// TIA Portal V18 export
// export: Created 2026-06-20T08:02:04.9898097Z, ExportSetting WithDefaults, DisplayName Totally Integrated Automation Portal, DisplayVersion V18, DisplayName TIA Portal Openness, DisplayVersion V18, DisplayName TIA Portal Version Control Interface, DisplayVersion V18, DisplayName STEP 7 Professional, DisplayVersion V18, DisplayName STEP 7 Safety, DisplayVersion V18, DisplayName WinCC Professional, DisplayVersion V18
ORGANIZATION_BLOCK "Main"   // OB1, LAD, ProgramCycle
TITLE = "Main Program Sweep (Cycle)"
{ S7_Optimized_Access := 'TRUE' }
VERSION : 0.1
// stored: AutoNumber true, IsIECCheckEnabled false, SetENOAutomatically false
   VAR_INPUT
      Initial_Call : Bool;   // Initial call of this OB
      Remanence : Bool;   // =True, if remanent data are available
   END_VAR
BEGIN

REGION Network 1: Clock 1Hz Edge Detection
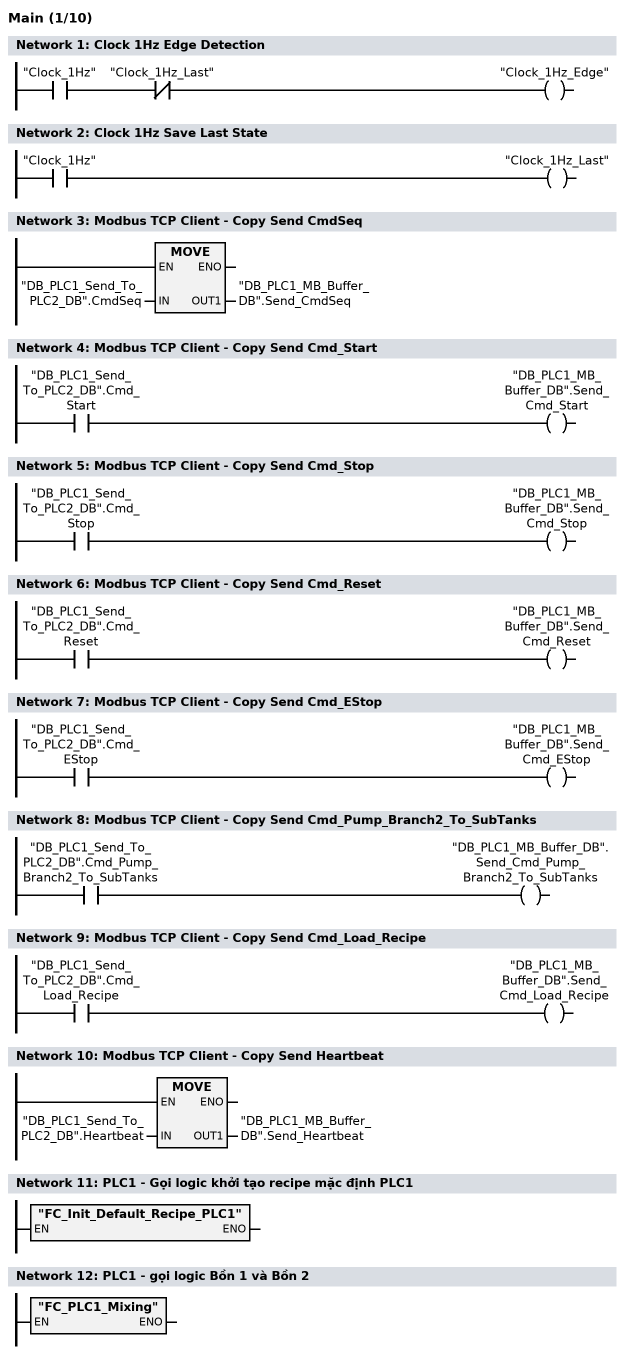
   RUNG wire#powerrail
      Contact( "Clock_1Hz" )
      I_Contact( "Clock_1Hz_Last" )
      Coil( "Clock_1Hz_Edge" )
   END_RUNG
   // the same network as SCL:
   "Clock_1Hz_Edge" := "Clock_1Hz" AND NOT "Clock_1Hz_Last";
END_REGION

REGION Network 2: Clock 1Hz Save Last State
   RUNG wire#powerrail
      Contact( "Clock_1Hz" )
      Coil( "Clock_1Hz_Last" )
   END_RUNG
   // the same network as SCL:
   "Clock_1Hz_Last" := "Clock_1Hz";
END_REGION

REGION Network 3: Modbus TCP Client - Copy Send CmdSeq
   RUNG wire#powerrail
      { S7_GenerateENO := "TRUE" } Move(in := "DB_PLC1_Send_To_PLC2_DB".CmdSeq, out1 => "DB_PLC1_MB_Buffer_DB".Send_CmdSeq)
   END_RUNG
   // the same network as SCL:
   "DB_PLC1_MB_Buffer_DB".Send_CmdSeq := "DB_PLC1_Send_To_PLC2_DB".CmdSeq;
END_REGION

REGION Network 4: Modbus TCP Client - Copy Send Cmd_Start
   RUNG wire#powerrail
      Contact( "DB_PLC1_Send_To_PLC2_DB".Cmd_Start )
      Coil( "DB_PLC1_MB_Buffer_DB".Send_Cmd_Start )
   END_RUNG
   // the same network as SCL:
   "DB_PLC1_MB_Buffer_DB".Send_Cmd_Start := "DB_PLC1_Send_To_PLC2_DB".Cmd_Start;
END_REGION

REGION Network 5: Modbus TCP Client - Copy Send Cmd_Stop
   RUNG wire#powerrail
      Contact( "DB_PLC1_Send_To_PLC2_DB".Cmd_Stop )
      Coil( "DB_PLC1_MB_Buffer_DB".Send_Cmd_Stop )
   END_RUNG
   // the same network as SCL:
   "DB_PLC1_MB_Buffer_DB".Send_Cmd_Stop := "DB_PLC1_Send_To_PLC2_DB".Cmd_Stop;
END_REGION

REGION Network 6: Modbus TCP Client - Copy Send Cmd_Reset
   RUNG wire#powerrail
      Contact( "DB_PLC1_Send_To_PLC2_DB".Cmd_Reset )
      Coil( "DB_PLC1_MB_Buffer_DB".Send_Cmd_Reset )
   END_RUNG
   // the same network as SCL:
   "DB_PLC1_MB_Buffer_DB".Send_Cmd_Reset := "DB_PLC1_Send_To_PLC2_DB".Cmd_Reset;
END_REGION

REGION Network 7: Modbus TCP Client - Copy Send Cmd_EStop
   RUNG wire#powerrail
      Contact( "DB_PLC1_Send_To_PLC2_DB".Cmd_EStop )
      Coil( "DB_PLC1_MB_Buffer_DB".Send_Cmd_EStop )
   END_RUNG
   // the same network as SCL:
   "DB_PLC1_MB_Buffer_DB".Send_Cmd_EStop := "DB_PLC1_Send_To_PLC2_DB".Cmd_EStop;
END_REGION

REGION Network 8: Modbus TCP Client - Copy Send Cmd_Pump_Branch2_To_SubTanks
   RUNG wire#powerrail
      Contact( "DB_PLC1_Send_To_PLC2_DB".Cmd_Pump_Branch2_To_SubTanks )
      Coil( "DB_PLC1_MB_Buffer_DB".Send_Cmd_Pump_Branch2_To_SubTanks )
   END_RUNG
   // the same network as SCL:
   "DB_PLC1_MB_Buffer_DB".Send_Cmd_Pump_Branch2_To_SubTanks := "DB_PLC1_Send_To_PLC2_DB".Cmd_Pump_Branch2_To_SubTanks;
END_REGION

REGION Network 9: Modbus TCP Client - Copy Send Cmd_Load_Recipe
   RUNG wire#powerrail
      Contact( "DB_PLC1_Send_To_PLC2_DB".Cmd_Load_Recipe )
      Coil( "DB_PLC1_MB_Buffer_DB".Send_Cmd_Load_Recipe )
   END_RUNG
   // the same network as SCL:
   "DB_PLC1_MB_Buffer_DB".Send_Cmd_Load_Recipe := "DB_PLC1_Send_To_PLC2_DB".Cmd_Load_Recipe;
END_REGION

REGION Network 10: Modbus TCP Client - Copy Send Heartbeat
   RUNG wire#powerrail
      { S7_GenerateENO := "TRUE" } Move(in := "DB_PLC1_Send_To_PLC2_DB".Heartbeat, out1 => "DB_PLC1_MB_Buffer_DB".Send_Heartbeat)
   END_RUNG
   // the same network as SCL:
   "DB_PLC1_MB_Buffer_DB".Send_Heartbeat := "DB_PLC1_Send_To_PLC2_DB".Heartbeat;
END_REGION

REGION Network 11: PLC1 - Gọi logic khởi tạo recipe mặc định PLC1
   RUNG wire#powerrail
      "FC_Init_Default_Recipe_PLC1"()
   END_RUNG
   // the same network as SCL:
   "FC_Init_Default_Recipe_PLC1"();
END_REGION

REGION Network 12: PLC1 - gọi logic Bồn 1 và Bồn 2
   RUNG wire#powerrail
      "FC_PLC1_Mixing"()
   END_RUNG
   // the same network as SCL:
   "FC_PLC1_Mixing"();
END_REGION

REGION Network 13: PLC1 - gọi logic bồn chứa và lọc thành phẩm
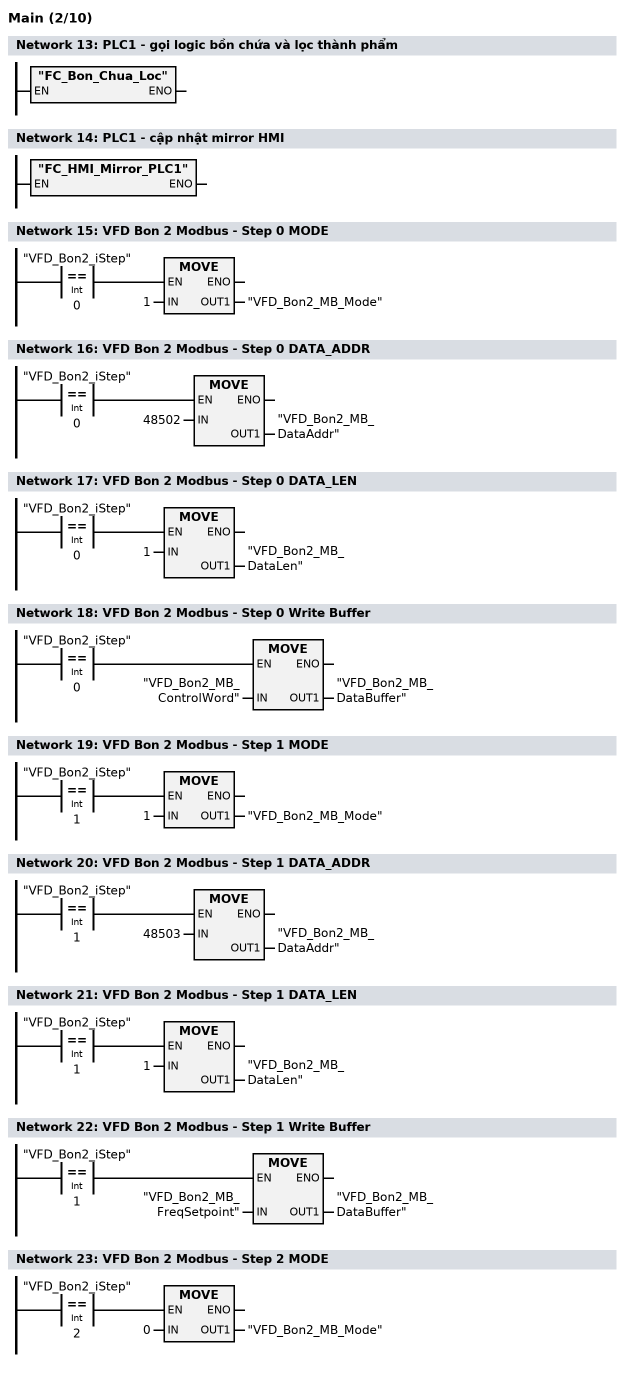
   RUNG wire#powerrail
      "FC_Bon_Chua_Loc"()
   END_RUNG
   // the same network as SCL:
   "FC_Bon_Chua_Loc"();
END_REGION

REGION Network 14: PLC1 - cập nhật mirror HMI
   RUNG wire#powerrail
      "FC_HMI_Mirror_PLC1"()
   END_RUNG
   // the same network as SCL:
   "FC_HMI_Mirror_PLC1"();
END_REGION

REGION Network 15: VFD Bon 2 Modbus - Step 0 MODE
   RUNG wire#powerrail
      { S7_Templates := "SrcType := Int" } EQ_Contact(in1 := "VFD_Bon2_iStep", in2 := 0)
      { S7_GenerateENO := "TRUE" } Move(in := 1, out1 => "VFD_Bon2_MB_Mode")
   END_RUNG
   // the same network as SCL:
   IF "VFD_Bon2_iStep" = 0 THEN "VFD_Bon2_MB_Mode" := 1; END_IF;
END_REGION

REGION Network 16: VFD Bon 2 Modbus - Step 0 DATA_ADDR
   RUNG wire#powerrail
      { S7_Templates := "SrcType := Int" } EQ_Contact(in1 := "VFD_Bon2_iStep", in2 := 0)
      { S7_GenerateENO := "TRUE" } Move(in := 48502, out1 => "VFD_Bon2_MB_DataAddr")
   END_RUNG
   // the same network as SCL:
   IF "VFD_Bon2_iStep" = 0 THEN "VFD_Bon2_MB_DataAddr" := 48502; END_IF;
END_REGION

REGION Network 17: VFD Bon 2 Modbus - Step 0 DATA_LEN
   RUNG wire#powerrail
      { S7_Templates := "SrcType := Int" } EQ_Contact(in1 := "VFD_Bon2_iStep", in2 := 0)
      { S7_GenerateENO := "TRUE" } Move(in := 1, out1 => "VFD_Bon2_MB_DataLen")
   END_RUNG
   // the same network as SCL:
   IF "VFD_Bon2_iStep" = 0 THEN "VFD_Bon2_MB_DataLen" := 1; END_IF;
END_REGION

REGION Network 18: VFD Bon 2 Modbus - Step 0 Write Buffer
   RUNG wire#powerrail
      { S7_Templates := "SrcType := Int" } EQ_Contact(in1 := "VFD_Bon2_iStep", in2 := 0)
      { S7_GenerateENO := "TRUE" } Move(in := "VFD_Bon2_MB_ControlWord", out1 => "VFD_Bon2_MB_DataBuffer")
   END_RUNG
   // the same network as SCL:
   IF "VFD_Bon2_iStep" = 0 THEN "VFD_Bon2_MB_DataBuffer" := "VFD_Bon2_MB_ControlWord"; END_IF;
END_REGION

REGION Network 19: VFD Bon 2 Modbus - Step 1 MODE
   RUNG wire#powerrail
      { S7_Templates := "SrcType := Int" } EQ_Contact(in1 := "VFD_Bon2_iStep", in2 := 1)
      { S7_GenerateENO := "TRUE" } Move(in := 1, out1 => "VFD_Bon2_MB_Mode")
   END_RUNG
   // the same network as SCL:
   IF "VFD_Bon2_iStep" = 1 THEN "VFD_Bon2_MB_Mode" := 1; END_IF;
END_REGION

REGION Network 20: VFD Bon 2 Modbus - Step 1 DATA_ADDR
   RUNG wire#powerrail
      { S7_Templates := "SrcType := Int" } EQ_Contact(in1 := "VFD_Bon2_iStep", in2 := 1)
      { S7_GenerateENO := "TRUE" } Move(in := 48503, out1 => "VFD_Bon2_MB_DataAddr")
   END_RUNG
   // the same network as SCL:
   IF "VFD_Bon2_iStep" = 1 THEN "VFD_Bon2_MB_DataAddr" := 48503; END_IF;
END_REGION

REGION Network 21: VFD Bon 2 Modbus - Step 1 DATA_LEN
   RUNG wire#powerrail
      { S7_Templates := "SrcType := Int" } EQ_Contact(in1 := "VFD_Bon2_iStep", in2 := 1)
      { S7_GenerateENO := "TRUE" } Move(in := 1, out1 => "VFD_Bon2_MB_DataLen")
   END_RUNG
   // the same network as SCL:
   IF "VFD_Bon2_iStep" = 1 THEN "VFD_Bon2_MB_DataLen" := 1; END_IF;
END_REGION

REGION Network 22: VFD Bon 2 Modbus - Step 1 Write Buffer
   RUNG wire#powerrail
      { S7_Templates := "SrcType := Int" } EQ_Contact(in1 := "VFD_Bon2_iStep", in2 := 1)
      { S7_GenerateENO := "TRUE" } Move(in := "VFD_Bon2_MB_FreqSetpoint", out1 => "VFD_Bon2_MB_DataBuffer")
   END_RUNG
   // the same network as SCL:
   IF "VFD_Bon2_iStep" = 1 THEN "VFD_Bon2_MB_DataBuffer" := "VFD_Bon2_MB_FreqSetpoint"; END_IF;
END_REGION

REGION Network 23: VFD Bon 2 Modbus - Step 2 MODE
   RUNG wire#powerrail
      { S7_Templates := "SrcType := Int" } EQ_Contact(in1 := "VFD_Bon2_iStep", in2 := 2)
      { S7_GenerateENO := "TRUE" } Move(in := 0, out1 => "VFD_Bon2_MB_Mode")
   END_RUNG
   // the same network as SCL:
   IF "VFD_Bon2_iStep" = 2 THEN "VFD_Bon2_MB_Mode" := 0; END_IF;
END_REGION

REGION Network 24: VFD Bon 2 Modbus - Step 2 DATA_ADDR
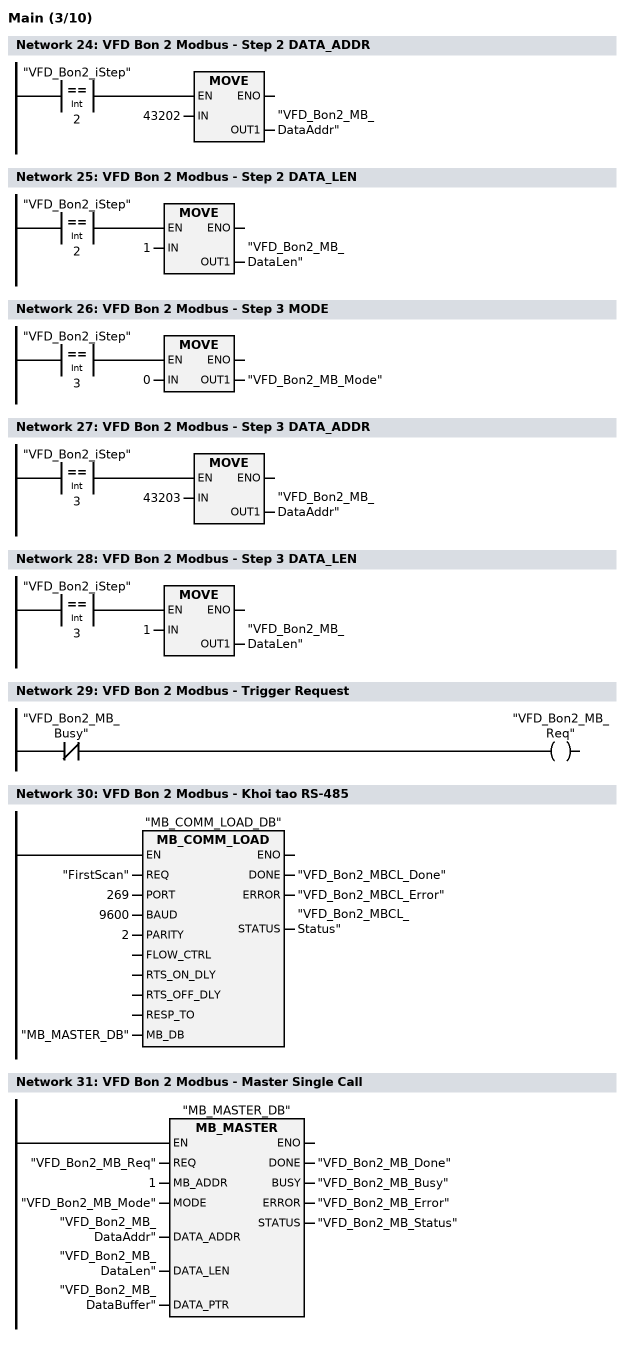
   RUNG wire#powerrail
      { S7_Templates := "SrcType := Int" } EQ_Contact(in1 := "VFD_Bon2_iStep", in2 := 2)
      { S7_GenerateENO := "TRUE" } Move(in := 43202, out1 => "VFD_Bon2_MB_DataAddr")
   END_RUNG
   // the same network as SCL:
   IF "VFD_Bon2_iStep" = 2 THEN "VFD_Bon2_MB_DataAddr" := 43202; END_IF;
END_REGION

REGION Network 25: VFD Bon 2 Modbus - Step 2 DATA_LEN
   RUNG wire#powerrail
      { S7_Templates := "SrcType := Int" } EQ_Contact(in1 := "VFD_Bon2_iStep", in2 := 2)
      { S7_GenerateENO := "TRUE" } Move(in := 1, out1 => "VFD_Bon2_MB_DataLen")
   END_RUNG
   // the same network as SCL:
   IF "VFD_Bon2_iStep" = 2 THEN "VFD_Bon2_MB_DataLen" := 1; END_IF;
END_REGION

REGION Network 26: VFD Bon 2 Modbus - Step 3 MODE
   RUNG wire#powerrail
      { S7_Templates := "SrcType := Int" } EQ_Contact(in1 := "VFD_Bon2_iStep", in2 := 3)
      { S7_GenerateENO := "TRUE" } Move(in := 0, out1 => "VFD_Bon2_MB_Mode")
   END_RUNG
   // the same network as SCL:
   IF "VFD_Bon2_iStep" = 3 THEN "VFD_Bon2_MB_Mode" := 0; END_IF;
END_REGION

REGION Network 27: VFD Bon 2 Modbus - Step 3 DATA_ADDR
   RUNG wire#powerrail
      { S7_Templates := "SrcType := Int" } EQ_Contact(in1 := "VFD_Bon2_iStep", in2 := 3)
      { S7_GenerateENO := "TRUE" } Move(in := 43203, out1 => "VFD_Bon2_MB_DataAddr")
   END_RUNG
   // the same network as SCL:
   IF "VFD_Bon2_iStep" = 3 THEN "VFD_Bon2_MB_DataAddr" := 43203; END_IF;
END_REGION

REGION Network 28: VFD Bon 2 Modbus - Step 3 DATA_LEN
   RUNG wire#powerrail
      { S7_Templates := "SrcType := Int" } EQ_Contact(in1 := "VFD_Bon2_iStep", in2 := 3)
      { S7_GenerateENO := "TRUE" } Move(in := 1, out1 => "VFD_Bon2_MB_DataLen")
   END_RUNG
   // the same network as SCL:
   IF "VFD_Bon2_iStep" = 3 THEN "VFD_Bon2_MB_DataLen" := 1; END_IF;
END_REGION

REGION Network 29: VFD Bon 2 Modbus - Trigger Request
   RUNG wire#powerrail
      I_Contact( "VFD_Bon2_MB_Busy" )
      Coil( "VFD_Bon2_MB_Req" )
   END_RUNG
   // the same network as SCL:
   "VFD_Bon2_MB_Req" := NOT "VFD_Bon2_MB_Busy";
END_REGION

REGION Network 30: VFD Bon 2 Modbus - Khoi tao RS-485
   RUNG wire#powerrail
      "MB_COMM_LOAD_DB".MB_COMM_LOAD(REQ := "FirstScan", PORT := 269, BAUD := 9600, PARITY := 2, FLOW_CTRL :=, RTS_ON_DLY :=, RTS_OFF_DLY :=, RESP_TO :=, MB_DB := "MB_MASTER_DB", DONE => "VFD_Bon2_MBCL_Done", ERROR => "VFD_Bon2_MBCL_Error", STATUS => "VFD_Bon2_MBCL_Status")
   END_RUNG
   // the same network as SCL:
   "MB_COMM_LOAD_DB"(REQ := "FirstScan",   // MB_COMM_LOAD
                     PORT := 269,
                     BAUD := 9600,
                     PARITY := 2,
                     MB_DB := "MB_MASTER_DB",
                     DONE => "VFD_Bon2_MBCL_Done",
                     ERROR => "VFD_Bon2_MBCL_Error",
                     STATUS => "VFD_Bon2_MBCL_Status");
END_REGION

REGION Network 31: VFD Bon 2 Modbus - Master Single Call
   RUNG wire#powerrail
      "MB_MASTER_DB".MB_MASTER(REQ := "VFD_Bon2_MB_Req", MB_ADDR := 1, MODE := "VFD_Bon2_MB_Mode", DATA_ADDR := "VFD_Bon2_MB_DataAddr", DATA_LEN := "VFD_Bon2_MB_DataLen", DATA_PTR := "VFD_Bon2_MB_DataBuffer", DONE => "VFD_Bon2_MB_Done", BUSY => "VFD_Bon2_MB_Busy", ERROR => "VFD_Bon2_MB_Error", STATUS => "VFD_Bon2_MB_Status")
   END_RUNG
   // the same network as SCL:
   "MB_MASTER_DB"(REQ := "VFD_Bon2_MB_Req",   // MB_MASTER
                  MB_ADDR := 1,
                  MODE := "VFD_Bon2_MB_Mode",
                  DATA_ADDR := "VFD_Bon2_MB_DataAddr",
                  DATA_LEN := "VFD_Bon2_MB_DataLen",
                  DATA_PTR := "VFD_Bon2_MB_DataBuffer",
                  DONE => "VFD_Bon2_MB_Done",
                  BUSY => "VFD_Bon2_MB_Busy",
                  ERROR => "VFD_Bon2_MB_Error",
                  STATUS => "VFD_Bon2_MB_Status");
END_REGION

REGION Network 32: VFD Bon 2 Modbus - Read Step 2 Buffer Copy
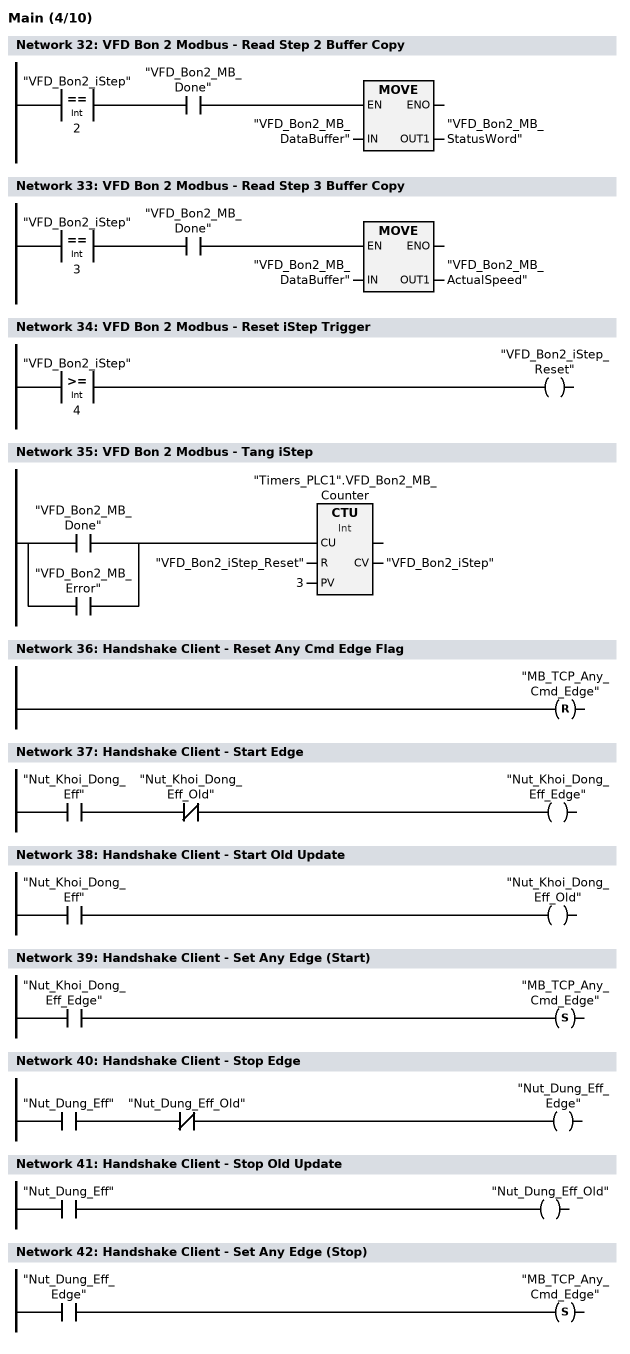
   RUNG wire#powerrail
      { S7_Templates := "SrcType := Int" } EQ_Contact(in1 := "VFD_Bon2_iStep", in2 := 2)
      Contact( "VFD_Bon2_MB_Done" )
      { S7_GenerateENO := "TRUE" } Move(in := "VFD_Bon2_MB_DataBuffer", out1 => "VFD_Bon2_MB_StatusWord")
   END_RUNG
   // the same network as SCL:
   IF ("VFD_Bon2_iStep" = 2) AND "VFD_Bon2_MB_Done" THEN
       "VFD_Bon2_MB_StatusWord" := "VFD_Bon2_MB_DataBuffer";
   END_IF;
END_REGION

REGION Network 33: VFD Bon 2 Modbus - Read Step 3 Buffer Copy
   RUNG wire#powerrail
      { S7_Templates := "SrcType := Int" } EQ_Contact(in1 := "VFD_Bon2_iStep", in2 := 3)
      Contact( "VFD_Bon2_MB_Done" )
      { S7_GenerateENO := "TRUE" } Move(in := "VFD_Bon2_MB_DataBuffer", out1 => "VFD_Bon2_MB_ActualSpeed")
   END_RUNG
   // the same network as SCL:
   IF ("VFD_Bon2_iStep" = 3) AND "VFD_Bon2_MB_Done" THEN
       "VFD_Bon2_MB_ActualSpeed" := "VFD_Bon2_MB_DataBuffer";
   END_IF;
END_REGION

REGION Network 34: VFD Bon 2 Modbus - Reset iStep Trigger
   RUNG wire#powerrail
      { S7_Templates := "SrcType := Int" } GE_Contact(in1 := "VFD_Bon2_iStep", in2 := 4)
      Coil( "VFD_Bon2_iStep_Reset" )
   END_RUNG
   // the same network as SCL:
   "VFD_Bon2_iStep_Reset" := "VFD_Bon2_iStep" >= 4;
END_REGION

REGION Network 35: VFD Bon 2 Modbus - Tang iStep
   RUNG wire#powerrail
      Contact( "VFD_Bon2_MB_Done" )
      wire#w1
      { S7_Templates := "value_type := Int" } "Timers_PLC1".VFD_Bon2_MB_Counter.CTU(r := "VFD_Bon2_iStep_Reset", pv := 3, cv => "VFD_Bon2_iStep")
   END_RUNG
   RUNG wire#powerrail
      Contact( "VFD_Bon2_MB_Error" )
   END_RUNG wire#w1
   // the same network as SCL:
   "Timers_PLC1".VFD_Bon2_MB_Counter.CTU(CU := "VFD_Bon2_MB_Done" OR "VFD_Bon2_MB_Error",
                           R := "VFD_Bon2_iStep_Reset",
                           PV := 3,
                           CV => "VFD_Bon2_iStep");
END_REGION

REGION Network 36: Handshake Client - Reset Any Cmd Edge Flag
   RUNG wire#powerrail
      R_Coil( "MB_TCP_Any_Cmd_Edge" )
   END_RUNG
   // the same network as SCL:
   "MB_TCP_Any_Cmd_Edge" := FALSE;
END_REGION

REGION Network 37: Handshake Client - Start Edge
   RUNG wire#powerrail
      Contact( "Nut_Khoi_Dong_Eff" )
      I_Contact( "Nut_Khoi_Dong_Eff_Old" )
      Coil( "Nut_Khoi_Dong_Eff_Edge" )
   END_RUNG
   // the same network as SCL:
   "Nut_Khoi_Dong_Eff_Edge" := "Nut_Khoi_Dong_Eff" AND NOT "Nut_Khoi_Dong_Eff_Old";
END_REGION

REGION Network 38: Handshake Client - Start Old Update
   RUNG wire#powerrail
      Contact( "Nut_Khoi_Dong_Eff" )
      Coil( "Nut_Khoi_Dong_Eff_Old" )
   END_RUNG
   // the same network as SCL:
   "Nut_Khoi_Dong_Eff_Old" := "Nut_Khoi_Dong_Eff";
END_REGION

REGION Network 39: Handshake Client - Set Any Edge (Start)
   RUNG wire#powerrail
      Contact( "Nut_Khoi_Dong_Eff_Edge" )
      S_Coil( "MB_TCP_Any_Cmd_Edge" )
   END_RUNG
   // the same network as SCL:
   IF "Nut_Khoi_Dong_Eff_Edge" THEN "MB_TCP_Any_Cmd_Edge" := TRUE; END_IF;
END_REGION

REGION Network 40: Handshake Client - Stop Edge
   RUNG wire#powerrail
      Contact( "Nut_Dung_Eff" )
      I_Contact( "Nut_Dung_Eff_Old" )
      Coil( "Nut_Dung_Eff_Edge" )
   END_RUNG
   // the same network as SCL:
   "Nut_Dung_Eff_Edge" := "Nut_Dung_Eff" AND NOT "Nut_Dung_Eff_Old";
END_REGION

REGION Network 41: Handshake Client - Stop Old Update
   RUNG wire#powerrail
      Contact( "Nut_Dung_Eff" )
      Coil( "Nut_Dung_Eff_Old" )
   END_RUNG
   // the same network as SCL:
   "Nut_Dung_Eff_Old" := "Nut_Dung_Eff";
END_REGION

REGION Network 42: Handshake Client - Set Any Edge (Stop)
   RUNG wire#powerrail
      Contact( "Nut_Dung_Eff_Edge" )
      S_Coil( "MB_TCP_Any_Cmd_Edge" )
   END_RUNG
   // the same network as SCL:
   IF "Nut_Dung_Eff_Edge" THEN "MB_TCP_Any_Cmd_Edge" := TRUE; END_IF;
END_REGION

REGION Network 43: Handshake Client - Reset Edge
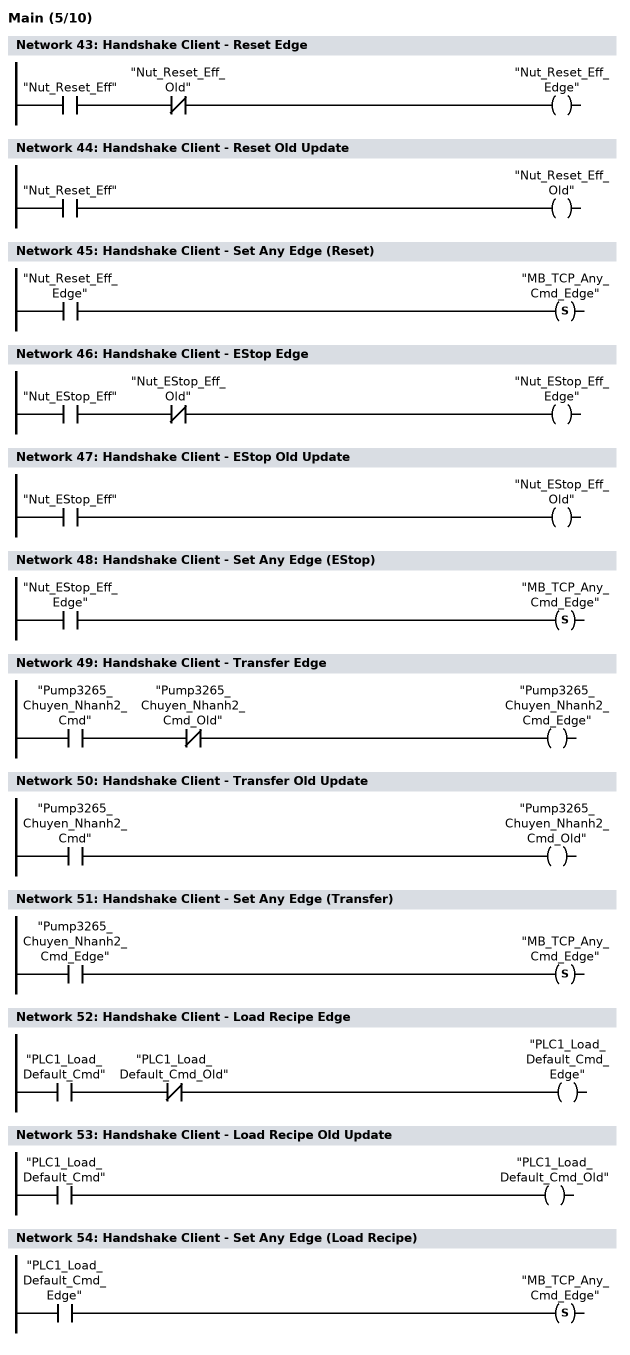
   RUNG wire#powerrail
      Contact( "Nut_Reset_Eff" )
      I_Contact( "Nut_Reset_Eff_Old" )
      Coil( "Nut_Reset_Eff_Edge" )
   END_RUNG
   // the same network as SCL:
   "Nut_Reset_Eff_Edge" := "Nut_Reset_Eff" AND NOT "Nut_Reset_Eff_Old";
END_REGION

REGION Network 44: Handshake Client - Reset Old Update
   RUNG wire#powerrail
      Contact( "Nut_Reset_Eff" )
      Coil( "Nut_Reset_Eff_Old" )
   END_RUNG
   // the same network as SCL:
   "Nut_Reset_Eff_Old" := "Nut_Reset_Eff";
END_REGION

REGION Network 45: Handshake Client - Set Any Edge (Reset)
   RUNG wire#powerrail
      Contact( "Nut_Reset_Eff_Edge" )
      S_Coil( "MB_TCP_Any_Cmd_Edge" )
   END_RUNG
   // the same network as SCL:
   IF "Nut_Reset_Eff_Edge" THEN "MB_TCP_Any_Cmd_Edge" := TRUE; END_IF;
END_REGION

REGION Network 46: Handshake Client - EStop Edge
   RUNG wire#powerrail
      Contact( "Nut_EStop_Eff" )
      I_Contact( "Nut_EStop_Eff_Old" )
      Coil( "Nut_EStop_Eff_Edge" )
   END_RUNG
   // the same network as SCL:
   "Nut_EStop_Eff_Edge" := "Nut_EStop_Eff" AND NOT "Nut_EStop_Eff_Old";
END_REGION

REGION Network 47: Handshake Client - EStop Old Update
   RUNG wire#powerrail
      Contact( "Nut_EStop_Eff" )
      Coil( "Nut_EStop_Eff_Old" )
   END_RUNG
   // the same network as SCL:
   "Nut_EStop_Eff_Old" := "Nut_EStop_Eff";
END_REGION

REGION Network 48: Handshake Client - Set Any Edge (EStop)
   RUNG wire#powerrail
      Contact( "Nut_EStop_Eff_Edge" )
      S_Coil( "MB_TCP_Any_Cmd_Edge" )
   END_RUNG
   // the same network as SCL:
   IF "Nut_EStop_Eff_Edge" THEN "MB_TCP_Any_Cmd_Edge" := TRUE; END_IF;
END_REGION

REGION Network 49: Handshake Client - Transfer Edge
   RUNG wire#powerrail
      Contact( "Pump3265_Chuyen_Nhanh2_Cmd" )
      I_Contact( "Pump3265_Chuyen_Nhanh2_Cmd_Old" )
      Coil( "Pump3265_Chuyen_Nhanh2_Cmd_Edge" )
   END_RUNG
   // the same network as SCL:
   "Pump3265_Chuyen_Nhanh2_Cmd_Edge" := "Pump3265_Chuyen_Nhanh2_Cmd" AND NOT "Pump3265_Chuyen_Nhanh2_Cmd_Old";
END_REGION

REGION Network 50: Handshake Client - Transfer Old Update
   RUNG wire#powerrail
      Contact( "Pump3265_Chuyen_Nhanh2_Cmd" )
      Coil( "Pump3265_Chuyen_Nhanh2_Cmd_Old" )
   END_RUNG
   // the same network as SCL:
   "Pump3265_Chuyen_Nhanh2_Cmd_Old" := "Pump3265_Chuyen_Nhanh2_Cmd";
END_REGION

REGION Network 51: Handshake Client - Set Any Edge (Transfer)
   RUNG wire#powerrail
      Contact( "Pump3265_Chuyen_Nhanh2_Cmd_Edge" )
      S_Coil( "MB_TCP_Any_Cmd_Edge" )
   END_RUNG
   // the same network as SCL:
   IF "Pump3265_Chuyen_Nhanh2_Cmd_Edge" THEN "MB_TCP_Any_Cmd_Edge" := TRUE; END_IF;
END_REGION

REGION Network 52: Handshake Client - Load Recipe Edge
   RUNG wire#powerrail
      Contact( "PLC1_Load_Default_Cmd" )
      I_Contact( "PLC1_Load_Default_Cmd_Old" )
      Coil( "PLC1_Load_Default_Cmd_Edge" )
   END_RUNG
   // the same network as SCL:
   "PLC1_Load_Default_Cmd_Edge" := "PLC1_Load_Default_Cmd" AND NOT "PLC1_Load_Default_Cmd_Old";
END_REGION

REGION Network 53: Handshake Client - Load Recipe Old Update
   RUNG wire#powerrail
      Contact( "PLC1_Load_Default_Cmd" )
      Coil( "PLC1_Load_Default_Cmd_Old" )
   END_RUNG
   // the same network as SCL:
   "PLC1_Load_Default_Cmd_Old" := "PLC1_Load_Default_Cmd";
END_REGION

REGION Network 54: Handshake Client - Set Any Edge (Load Recipe)
   RUNG wire#powerrail
      Contact( "PLC1_Load_Default_Cmd_Edge" )
      S_Coil( "MB_TCP_Any_Cmd_Edge" )
   END_RUNG
   // the same network as SCL:
   IF "PLC1_Load_Default_Cmd_Edge" THEN "MB_TCP_Any_Cmd_Edge" := TRUE; END_IF;
END_REGION

REGION Network 55: Handshake Client - Latch Start
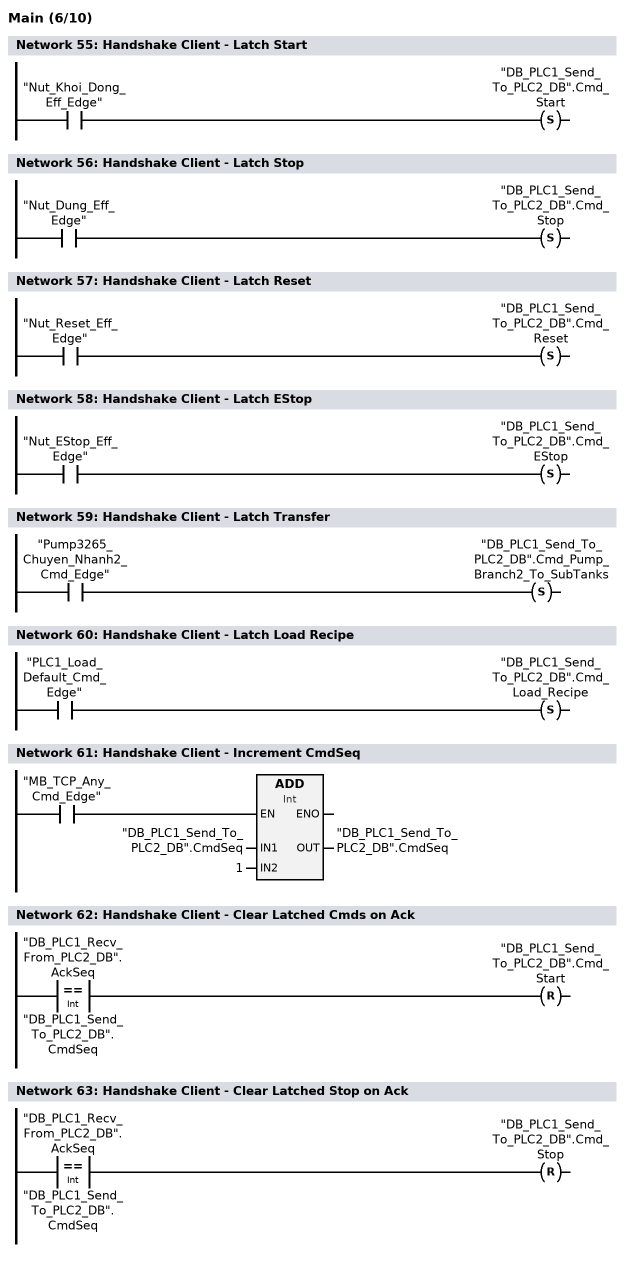
   RUNG wire#powerrail
      Contact( "Nut_Khoi_Dong_Eff_Edge" )
      S_Coil( "DB_PLC1_Send_To_PLC2_DB".Cmd_Start )
   END_RUNG
   // the same network as SCL:
   IF "Nut_Khoi_Dong_Eff_Edge" THEN "DB_PLC1_Send_To_PLC2_DB".Cmd_Start := TRUE; END_IF;
END_REGION

REGION Network 56: Handshake Client - Latch Stop
   RUNG wire#powerrail
      Contact( "Nut_Dung_Eff_Edge" )
      S_Coil( "DB_PLC1_Send_To_PLC2_DB".Cmd_Stop )
   END_RUNG
   // the same network as SCL:
   IF "Nut_Dung_Eff_Edge" THEN "DB_PLC1_Send_To_PLC2_DB".Cmd_Stop := TRUE; END_IF;
END_REGION

REGION Network 57: Handshake Client - Latch Reset
   RUNG wire#powerrail
      Contact( "Nut_Reset_Eff_Edge" )
      S_Coil( "DB_PLC1_Send_To_PLC2_DB".Cmd_Reset )
   END_RUNG
   // the same network as SCL:
   IF "Nut_Reset_Eff_Edge" THEN "DB_PLC1_Send_To_PLC2_DB".Cmd_Reset := TRUE; END_IF;
END_REGION

REGION Network 58: Handshake Client - Latch EStop
   RUNG wire#powerrail
      Contact( "Nut_EStop_Eff_Edge" )
      S_Coil( "DB_PLC1_Send_To_PLC2_DB".Cmd_EStop )
   END_RUNG
   // the same network as SCL:
   IF "Nut_EStop_Eff_Edge" THEN "DB_PLC1_Send_To_PLC2_DB".Cmd_EStop := TRUE; END_IF;
END_REGION

REGION Network 59: Handshake Client - Latch Transfer
   RUNG wire#powerrail
      Contact( "Pump3265_Chuyen_Nhanh2_Cmd_Edge" )
      S_Coil( "DB_PLC1_Send_To_PLC2_DB".Cmd_Pump_Branch2_To_SubTanks )
   END_RUNG
   // the same network as SCL:
   IF "Pump3265_Chuyen_Nhanh2_Cmd_Edge" THEN
       "DB_PLC1_Send_To_PLC2_DB".Cmd_Pump_Branch2_To_SubTanks := TRUE;
   END_IF;
END_REGION

REGION Network 60: Handshake Client - Latch Load Recipe
   RUNG wire#powerrail
      Contact( "PLC1_Load_Default_Cmd_Edge" )
      S_Coil( "DB_PLC1_Send_To_PLC2_DB".Cmd_Load_Recipe )
   END_RUNG
   // the same network as SCL:
   IF "PLC1_Load_Default_Cmd_Edge" THEN "DB_PLC1_Send_To_PLC2_DB".Cmd_Load_Recipe := TRUE; END_IF;
END_REGION

REGION Network 61: Handshake Client - Increment CmdSeq
   RUNG wire#powerrail
      Contact( "MB_TCP_Any_Cmd_Edge" )
      { S7_Templates := "SrcType := Int"; S7_GenerateENO := "TRUE" } Add(in1 := "DB_PLC1_Send_To_PLC2_DB".CmdSeq, in2 := 1, out => "DB_PLC1_Send_To_PLC2_DB".CmdSeq)
   END_RUNG
   // the same network as SCL:
   IF "MB_TCP_Any_Cmd_Edge" THEN
       "DB_PLC1_Send_To_PLC2_DB".CmdSeq := "DB_PLC1_Send_To_PLC2_DB".CmdSeq + 1;
   END_IF;
END_REGION

REGION Network 62: Handshake Client - Clear Latched Cmds on Ack
   RUNG wire#powerrail
      { S7_Templates := "SrcType := Int" } EQ_Contact(in1 := "DB_PLC1_Recv_From_PLC2_DB".AckSeq, in2 := "DB_PLC1_Send_To_PLC2_DB".CmdSeq)
      R_Coil( "DB_PLC1_Send_To_PLC2_DB".Cmd_Start )
   END_RUNG
   // the same network as SCL:
   IF "DB_PLC1_Recv_From_PLC2_DB".AckSeq = "DB_PLC1_Send_To_PLC2_DB".CmdSeq THEN
       "DB_PLC1_Send_To_PLC2_DB".Cmd_Start := FALSE;
   END_IF;
END_REGION

REGION Network 63: Handshake Client - Clear Latched Stop on Ack
   RUNG wire#powerrail
      { S7_Templates := "SrcType := Int" } EQ_Contact(in1 := "DB_PLC1_Recv_From_PLC2_DB".AckSeq, in2 := "DB_PLC1_Send_To_PLC2_DB".CmdSeq)
      R_Coil( "DB_PLC1_Send_To_PLC2_DB".Cmd_Stop )
   END_RUNG
   // the same network as SCL:
   IF "DB_PLC1_Recv_From_PLC2_DB".AckSeq = "DB_PLC1_Send_To_PLC2_DB".CmdSeq THEN
       "DB_PLC1_Send_To_PLC2_DB".Cmd_Stop := FALSE;
   END_IF;
END_REGION

REGION Network 64: Handshake Client - Clear Latched Reset on Ack
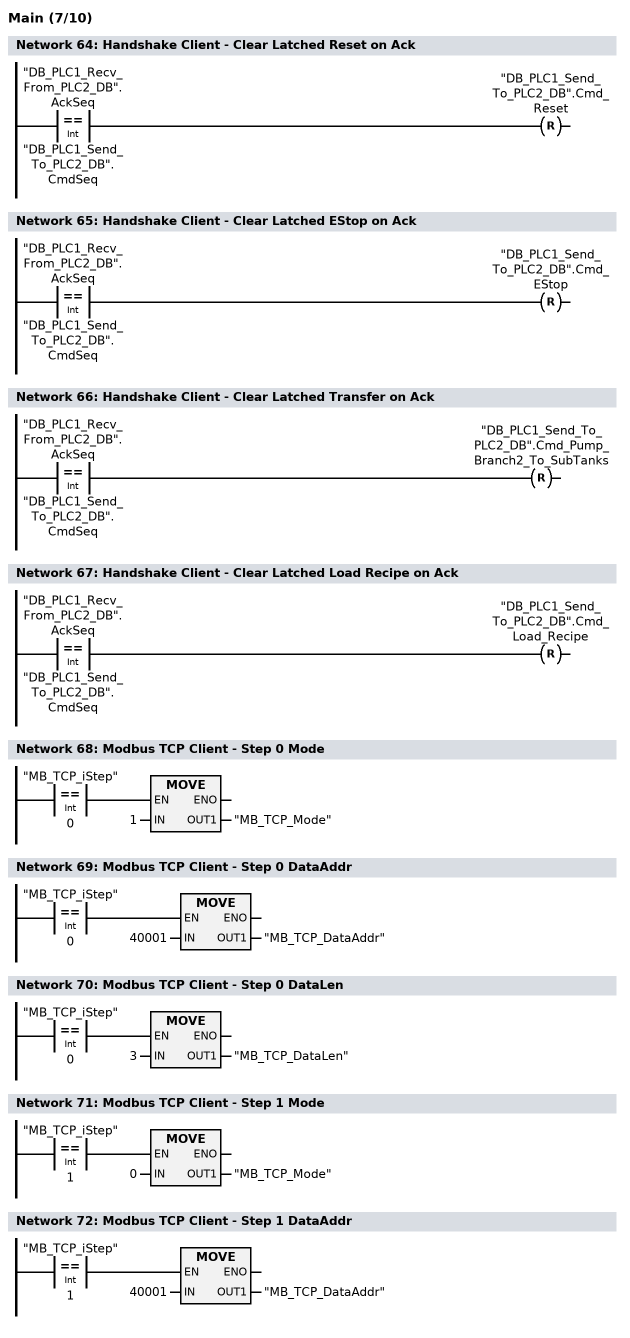
   RUNG wire#powerrail
      { S7_Templates := "SrcType := Int" } EQ_Contact(in1 := "DB_PLC1_Recv_From_PLC2_DB".AckSeq, in2 := "DB_PLC1_Send_To_PLC2_DB".CmdSeq)
      R_Coil( "DB_PLC1_Send_To_PLC2_DB".Cmd_Reset )
   END_RUNG
   // the same network as SCL:
   IF "DB_PLC1_Recv_From_PLC2_DB".AckSeq = "DB_PLC1_Send_To_PLC2_DB".CmdSeq THEN
       "DB_PLC1_Send_To_PLC2_DB".Cmd_Reset := FALSE;
   END_IF;
END_REGION

REGION Network 65: Handshake Client - Clear Latched EStop on Ack
   RUNG wire#powerrail
      { S7_Templates := "SrcType := Int" } EQ_Contact(in1 := "DB_PLC1_Recv_From_PLC2_DB".AckSeq, in2 := "DB_PLC1_Send_To_PLC2_DB".CmdSeq)
      R_Coil( "DB_PLC1_Send_To_PLC2_DB".Cmd_EStop )
   END_RUNG
   // the same network as SCL:
   IF "DB_PLC1_Recv_From_PLC2_DB".AckSeq = "DB_PLC1_Send_To_PLC2_DB".CmdSeq THEN
       "DB_PLC1_Send_To_PLC2_DB".Cmd_EStop := FALSE;
   END_IF;
END_REGION

REGION Network 66: Handshake Client - Clear Latched Transfer on Ack
   RUNG wire#powerrail
      { S7_Templates := "SrcType := Int" } EQ_Contact(in1 := "DB_PLC1_Recv_From_PLC2_DB".AckSeq, in2 := "DB_PLC1_Send_To_PLC2_DB".CmdSeq)
      R_Coil( "DB_PLC1_Send_To_PLC2_DB".Cmd_Pump_Branch2_To_SubTanks )
   END_RUNG
   // the same network as SCL:
   IF "DB_PLC1_Recv_From_PLC2_DB".AckSeq = "DB_PLC1_Send_To_PLC2_DB".CmdSeq THEN
       "DB_PLC1_Send_To_PLC2_DB".Cmd_Pump_Branch2_To_SubTanks := FALSE;
   END_IF;
END_REGION

REGION Network 67: Handshake Client - Clear Latched Load Recipe on Ack
   RUNG wire#powerrail
      { S7_Templates := "SrcType := Int" } EQ_Contact(in1 := "DB_PLC1_Recv_From_PLC2_DB".AckSeq, in2 := "DB_PLC1_Send_To_PLC2_DB".CmdSeq)
      R_Coil( "DB_PLC1_Send_To_PLC2_DB".Cmd_Load_Recipe )
   END_RUNG
   // the same network as SCL:
   IF "DB_PLC1_Recv_From_PLC2_DB".AckSeq = "DB_PLC1_Send_To_PLC2_DB".CmdSeq THEN
       "DB_PLC1_Send_To_PLC2_DB".Cmd_Load_Recipe := FALSE;
   END_IF;
END_REGION

REGION Network 68: Modbus TCP Client - Step 0 Mode
   RUNG wire#powerrail
      { S7_Templates := "SrcType := Int" } EQ_Contact(in1 := "MB_TCP_iStep", in2 := 0)
      { S7_GenerateENO := "TRUE" } Move(in := 1, out1 => "MB_TCP_Mode")
   END_RUNG
   // the same network as SCL:
   IF "MB_TCP_iStep" = 0 THEN "MB_TCP_Mode" := 1; END_IF;
END_REGION

REGION Network 69: Modbus TCP Client - Step 0 DataAddr
   RUNG wire#powerrail
      { S7_Templates := "SrcType := Int" } EQ_Contact(in1 := "MB_TCP_iStep", in2 := 0)
      { S7_GenerateENO := "TRUE" } Move(in := 40001, out1 => "MB_TCP_DataAddr")
   END_RUNG
   // the same network as SCL:
   IF "MB_TCP_iStep" = 0 THEN "MB_TCP_DataAddr" := 40001; END_IF;
END_REGION

REGION Network 70: Modbus TCP Client - Step 0 DataLen
   RUNG wire#powerrail
      { S7_Templates := "SrcType := Int" } EQ_Contact(in1 := "MB_TCP_iStep", in2 := 0)
      { S7_GenerateENO := "TRUE" } Move(in := 3, out1 => "MB_TCP_DataLen")
   END_RUNG
   // the same network as SCL:
   IF "MB_TCP_iStep" = 0 THEN "MB_TCP_DataLen" := 3; END_IF;
END_REGION

REGION Network 71: Modbus TCP Client - Step 1 Mode
   RUNG wire#powerrail
      { S7_Templates := "SrcType := Int" } EQ_Contact(in1 := "MB_TCP_iStep", in2 := 1)
      { S7_GenerateENO := "TRUE" } Move(in := 0, out1 => "MB_TCP_Mode")
   END_RUNG
   // the same network as SCL:
   IF "MB_TCP_iStep" = 1 THEN "MB_TCP_Mode" := 0; END_IF;
END_REGION

REGION Network 72: Modbus TCP Client - Step 1 DataAddr
   RUNG wire#powerrail
      { S7_Templates := "SrcType := Int" } EQ_Contact(in1 := "MB_TCP_iStep", in2 := 1)
      { S7_GenerateENO := "TRUE" } Move(in := 40001, out1 => "MB_TCP_DataAddr")
   END_RUNG
   // the same network as SCL:
   IF "MB_TCP_iStep" = 1 THEN "MB_TCP_DataAddr" := 40001; END_IF;
END_REGION

REGION Network 73: Modbus TCP Client - Step 1 DataLen
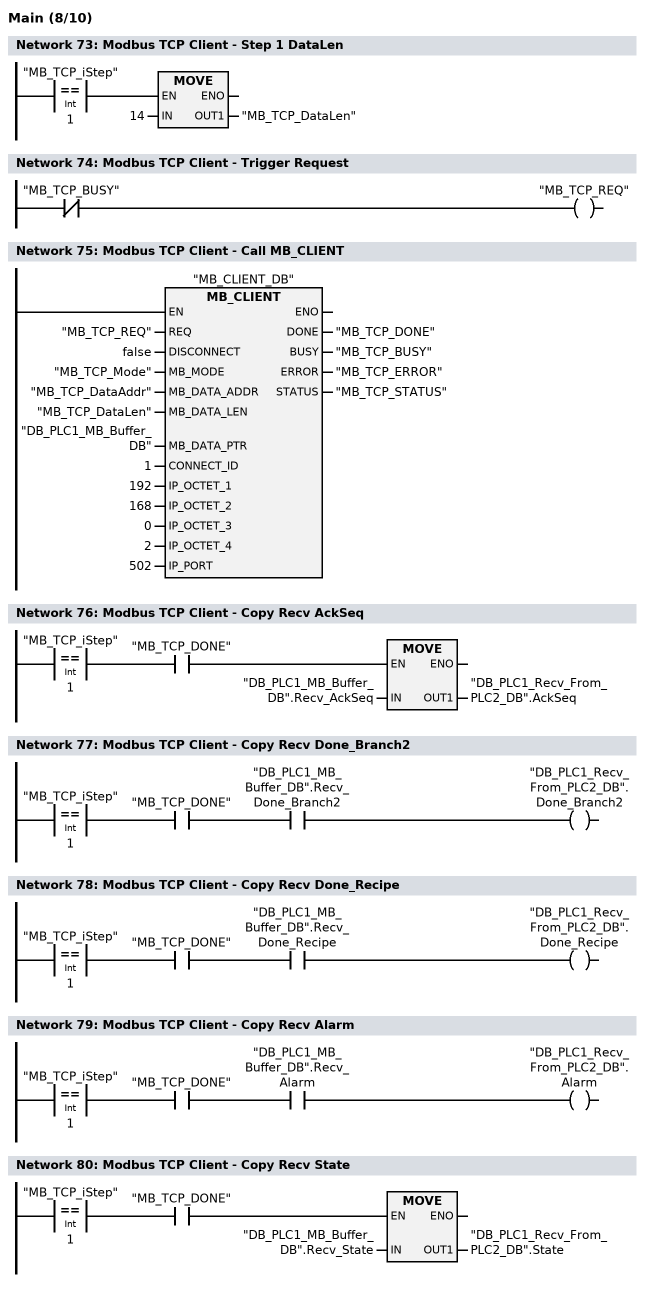
   RUNG wire#powerrail
      { S7_Templates := "SrcType := Int" } EQ_Contact(in1 := "MB_TCP_iStep", in2 := 1)
      { S7_GenerateENO := "TRUE" } Move(in := 14, out1 => "MB_TCP_DataLen")
   END_RUNG
   // the same network as SCL:
   IF "MB_TCP_iStep" = 1 THEN "MB_TCP_DataLen" := 14; END_IF;
END_REGION

REGION Network 74: Modbus TCP Client - Trigger Request
   RUNG wire#powerrail
      I_Contact( "MB_TCP_BUSY" )
      Coil( "MB_TCP_REQ" )
   END_RUNG
   // the same network as SCL:
   "MB_TCP_REQ" := NOT "MB_TCP_BUSY";
END_REGION

REGION Network 75: Modbus TCP Client - Call MB_CLIENT
   RUNG wire#powerrail
      { S7_Templates := "[card1200 := 1, card1500 := 0]" } "MB_CLIENT_DB".MB_CLIENT(REQ := "MB_TCP_REQ", DISCONNECT := false, MB_MODE := "MB_TCP_Mode", MB_DATA_ADDR := "MB_TCP_DataAddr", MB_DATA_LEN := "MB_TCP_DataLen", MB_DATA_PTR := "DB_PLC1_MB_Buffer_DB", CONNECT_ID := 1, IP_OCTET_1 := 192, IP_OCTET_2 := 168, IP_OCTET_3 := 0, IP_OCTET_4 := 2, IP_PORT := 502, DONE => "MB_TCP_DONE", BUSY => "MB_TCP_BUSY", ERROR => "MB_TCP_ERROR", STATUS => "MB_TCP_STATUS")
   END_RUNG
   // the same network as SCL:
   "MB_CLIENT_DB"(REQ := "MB_TCP_REQ",   // MB_CLIENT
                  DISCONNECT := false,
                  MB_MODE := "MB_TCP_Mode",
                  MB_DATA_ADDR := "MB_TCP_DataAddr",
                  MB_DATA_LEN := "MB_TCP_DataLen",
                  MB_DATA_PTR := "DB_PLC1_MB_Buffer_DB",
                  CONNECT_ID := 1,
                  IP_OCTET_1 := 192,
                  IP_OCTET_2 := 168,
                  IP_OCTET_3 := 0,
                  IP_OCTET_4 := 2,
                  IP_PORT := 502,
                  DONE => "MB_TCP_DONE",
                  BUSY => "MB_TCP_BUSY",
                  ERROR => "MB_TCP_ERROR",
                  STATUS => "MB_TCP_STATUS");
END_REGION

REGION Network 76: Modbus TCP Client - Copy Recv AckSeq
   RUNG wire#powerrail
      { S7_Templates := "SrcType := Int" } EQ_Contact(in1 := "MB_TCP_iStep", in2 := 1)
      Contact( "MB_TCP_DONE" )
      { S7_GenerateENO := "TRUE" } Move(in := "DB_PLC1_MB_Buffer_DB".Recv_AckSeq, out1 => "DB_PLC1_Recv_From_PLC2_DB".AckSeq)
   END_RUNG
   // the same network as SCL:
   IF ("MB_TCP_iStep" = 1) AND "MB_TCP_DONE" THEN
       "DB_PLC1_Recv_From_PLC2_DB".AckSeq := "DB_PLC1_MB_Buffer_DB".Recv_AckSeq;
   END_IF;
END_REGION

REGION Network 77: Modbus TCP Client - Copy Recv Done_Branch2
   RUNG wire#powerrail
      { S7_Templates := "SrcType := Int" } EQ_Contact(in1 := "MB_TCP_iStep", in2 := 1)
      Contact( "MB_TCP_DONE" )
      Contact( "DB_PLC1_MB_Buffer_DB".Recv_Done_Branch2 )
      Coil( "DB_PLC1_Recv_From_PLC2_DB".Done_Branch2 )
   END_RUNG
   // the same network as SCL:
   "DB_PLC1_Recv_From_PLC2_DB".Done_Branch2 := ("MB_TCP_iStep" = 1) AND "MB_TCP_DONE" AND "DB_PLC1_MB_Buffer_DB".Recv_Done_Branch2;
END_REGION

REGION Network 78: Modbus TCP Client - Copy Recv Done_Recipe
   RUNG wire#powerrail
      { S7_Templates := "SrcType := Int" } EQ_Contact(in1 := "MB_TCP_iStep", in2 := 1)
      Contact( "MB_TCP_DONE" )
      Contact( "DB_PLC1_MB_Buffer_DB".Recv_Done_Recipe )
      Coil( "DB_PLC1_Recv_From_PLC2_DB".Done_Recipe )
   END_RUNG
   // the same network as SCL:
   "DB_PLC1_Recv_From_PLC2_DB".Done_Recipe := ("MB_TCP_iStep" = 1) AND "MB_TCP_DONE" AND "DB_PLC1_MB_Buffer_DB".Recv_Done_Recipe;
END_REGION

REGION Network 79: Modbus TCP Client - Copy Recv Alarm
   RUNG wire#powerrail
      { S7_Templates := "SrcType := Int" } EQ_Contact(in1 := "MB_TCP_iStep", in2 := 1)
      Contact( "MB_TCP_DONE" )
      Contact( "DB_PLC1_MB_Buffer_DB".Recv_Alarm )
      Coil( "DB_PLC1_Recv_From_PLC2_DB".Alarm )
   END_RUNG
   // the same network as SCL:
   "DB_PLC1_Recv_From_PLC2_DB".Alarm := ("MB_TCP_iStep" = 1) AND "MB_TCP_DONE" AND "DB_PLC1_MB_Buffer_DB".Recv_Alarm;
END_REGION

REGION Network 80: Modbus TCP Client - Copy Recv State
   RUNG wire#powerrail
      { S7_Templates := "SrcType := Int" } EQ_Contact(in1 := "MB_TCP_iStep", in2 := 1)
      Contact( "MB_TCP_DONE" )
      { S7_GenerateENO := "TRUE" } Move(in := "DB_PLC1_MB_Buffer_DB".Recv_State, out1 => "DB_PLC1_Recv_From_PLC2_DB".State)
   END_RUNG
   // the same network as SCL:
   IF ("MB_TCP_iStep" = 1) AND "MB_TCP_DONE" THEN
       "DB_PLC1_Recv_From_PLC2_DB".State := "DB_PLC1_MB_Buffer_DB".Recv_State;
   END_IF;
END_REGION

REGION Network 81: Modbus TCP Client - Copy Recv PID_Bon4_SP
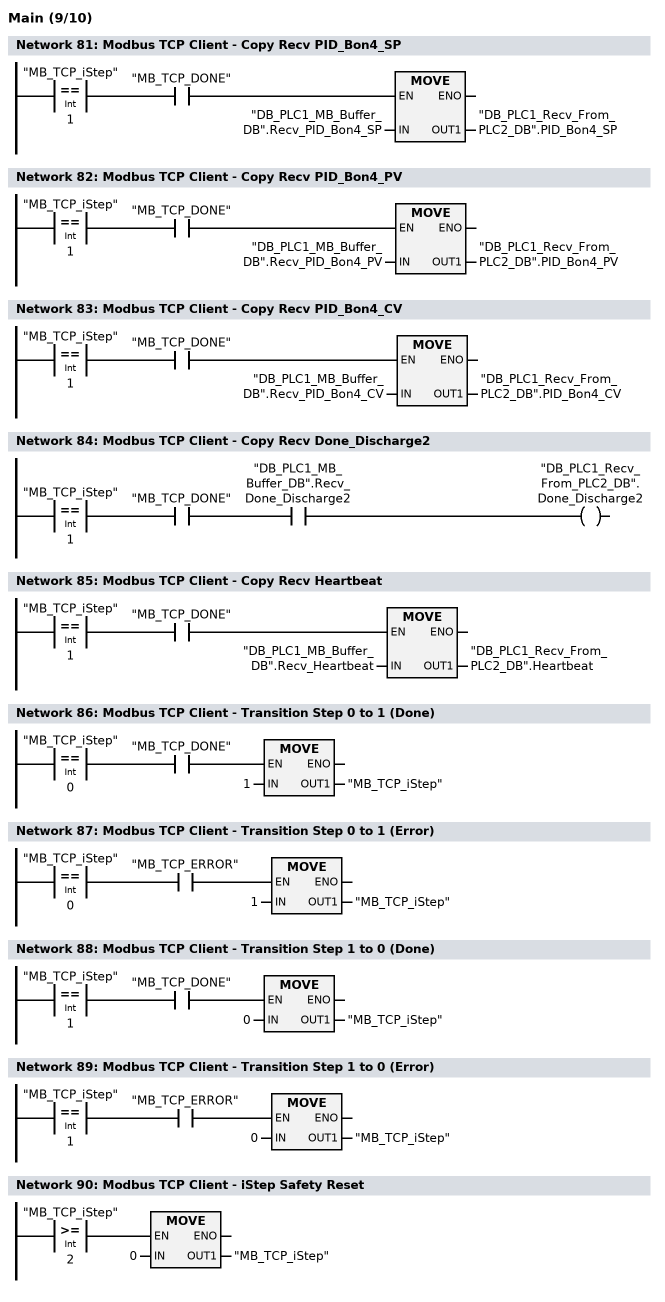
   RUNG wire#powerrail
      { S7_Templates := "SrcType := Int" } EQ_Contact(in1 := "MB_TCP_iStep", in2 := 1)
      Contact( "MB_TCP_DONE" )
      { S7_GenerateENO := "TRUE" } Move(in := "DB_PLC1_MB_Buffer_DB".Recv_PID_Bon4_SP, out1 => "DB_PLC1_Recv_From_PLC2_DB".PID_Bon4_SP)
   END_RUNG
   // the same network as SCL:
   IF ("MB_TCP_iStep" = 1) AND "MB_TCP_DONE" THEN
       "DB_PLC1_Recv_From_PLC2_DB".PID_Bon4_SP := "DB_PLC1_MB_Buffer_DB".Recv_PID_Bon4_SP;
   END_IF;
END_REGION

REGION Network 82: Modbus TCP Client - Copy Recv PID_Bon4_PV
   RUNG wire#powerrail
      { S7_Templates := "SrcType := Int" } EQ_Contact(in1 := "MB_TCP_iStep", in2 := 1)
      Contact( "MB_TCP_DONE" )
      { S7_GenerateENO := "TRUE" } Move(in := "DB_PLC1_MB_Buffer_DB".Recv_PID_Bon4_PV, out1 => "DB_PLC1_Recv_From_PLC2_DB".PID_Bon4_PV)
   END_RUNG
   // the same network as SCL:
   IF ("MB_TCP_iStep" = 1) AND "MB_TCP_DONE" THEN
       "DB_PLC1_Recv_From_PLC2_DB".PID_Bon4_PV := "DB_PLC1_MB_Buffer_DB".Recv_PID_Bon4_PV;
   END_IF;
END_REGION

REGION Network 83: Modbus TCP Client - Copy Recv PID_Bon4_CV
   RUNG wire#powerrail
      { S7_Templates := "SrcType := Int" } EQ_Contact(in1 := "MB_TCP_iStep", in2 := 1)
      Contact( "MB_TCP_DONE" )
      { S7_GenerateENO := "TRUE" } Move(in := "DB_PLC1_MB_Buffer_DB".Recv_PID_Bon4_CV, out1 => "DB_PLC1_Recv_From_PLC2_DB".PID_Bon4_CV)
   END_RUNG
   // the same network as SCL:
   IF ("MB_TCP_iStep" = 1) AND "MB_TCP_DONE" THEN
       "DB_PLC1_Recv_From_PLC2_DB".PID_Bon4_CV := "DB_PLC1_MB_Buffer_DB".Recv_PID_Bon4_CV;
   END_IF;
END_REGION

REGION Network 84: Modbus TCP Client - Copy Recv Done_Discharge2
   RUNG wire#powerrail
      { S7_Templates := "SrcType := Int" } EQ_Contact(in1 := "MB_TCP_iStep", in2 := 1)
      Contact( "MB_TCP_DONE" )
      Contact( "DB_PLC1_MB_Buffer_DB".Recv_Done_Discharge2 )
      Coil( "DB_PLC1_Recv_From_PLC2_DB".Done_Discharge2 )
   END_RUNG
   // the same network as SCL:
   "DB_PLC1_Recv_From_PLC2_DB".Done_Discharge2 := ("MB_TCP_iStep" = 1) AND "MB_TCP_DONE" AND "DB_PLC1_MB_Buffer_DB".Recv_Done_Discharge2;
END_REGION

REGION Network 85: Modbus TCP Client - Copy Recv Heartbeat
   RUNG wire#powerrail
      { S7_Templates := "SrcType := Int" } EQ_Contact(in1 := "MB_TCP_iStep", in2 := 1)
      Contact( "MB_TCP_DONE" )
      { S7_GenerateENO := "TRUE" } Move(in := "DB_PLC1_MB_Buffer_DB".Recv_Heartbeat, out1 => "DB_PLC1_Recv_From_PLC2_DB".Heartbeat)
   END_RUNG
   // the same network as SCL:
   IF ("MB_TCP_iStep" = 1) AND "MB_TCP_DONE" THEN
       "DB_PLC1_Recv_From_PLC2_DB".Heartbeat := "DB_PLC1_MB_Buffer_DB".Recv_Heartbeat;
   END_IF;
END_REGION

REGION Network 86: Modbus TCP Client - Transition Step 0 to 1 (Done)
   RUNG wire#powerrail
      { S7_Templates := "SrcType := Int" } EQ_Contact(in1 := "MB_TCP_iStep", in2 := 0)
      Contact( "MB_TCP_DONE" )
      { S7_GenerateENO := "TRUE" } Move(in := 1, out1 => "MB_TCP_iStep")
   END_RUNG
   // the same network as SCL:
   IF ("MB_TCP_iStep" = 0) AND "MB_TCP_DONE" THEN "MB_TCP_iStep" := 1; END_IF;
END_REGION

REGION Network 87: Modbus TCP Client - Transition Step 0 to 1 (Error)
   RUNG wire#powerrail
      { S7_Templates := "SrcType := Int" } EQ_Contact(in1 := "MB_TCP_iStep", in2 := 0)
      Contact( "MB_TCP_ERROR" )
      { S7_GenerateENO := "TRUE" } Move(in := 1, out1 => "MB_TCP_iStep")
   END_RUNG
   // the same network as SCL:
   IF ("MB_TCP_iStep" = 0) AND "MB_TCP_ERROR" THEN "MB_TCP_iStep" := 1; END_IF;
END_REGION

REGION Network 88: Modbus TCP Client - Transition Step 1 to 0 (Done)
   RUNG wire#powerrail
      { S7_Templates := "SrcType := Int" } EQ_Contact(in1 := "MB_TCP_iStep", in2 := 1)
      Contact( "MB_TCP_DONE" )
      { S7_GenerateENO := "TRUE" } Move(in := 0, out1 => "MB_TCP_iStep")
   END_RUNG
   // the same network as SCL:
   IF ("MB_TCP_iStep" = 1) AND "MB_TCP_DONE" THEN "MB_TCP_iStep" := 0; END_IF;
END_REGION

REGION Network 89: Modbus TCP Client - Transition Step 1 to 0 (Error)
   RUNG wire#powerrail
      { S7_Templates := "SrcType := Int" } EQ_Contact(in1 := "MB_TCP_iStep", in2 := 1)
      Contact( "MB_TCP_ERROR" )
      { S7_GenerateENO := "TRUE" } Move(in := 0, out1 => "MB_TCP_iStep")
   END_RUNG
   // the same network as SCL:
   IF ("MB_TCP_iStep" = 1) AND "MB_TCP_ERROR" THEN "MB_TCP_iStep" := 0; END_IF;
END_REGION

REGION Network 90: Modbus TCP Client - iStep Safety Reset
   RUNG wire#powerrail
      { S7_Templates := "SrcType := Int" } GE_Contact(in1 := "MB_TCP_iStep", in2 := 2)
      { S7_GenerateENO := "TRUE" } Move(in := 0, out1 => "MB_TCP_iStep")
   END_RUNG
   // the same network as SCL:
   IF "MB_TCP_iStep" >= 2 THEN "MB_TCP_iStep" := 0; END_IF;
END_REGION

REGION Network 91: Modbus TCP Client - Increment Heartbeat
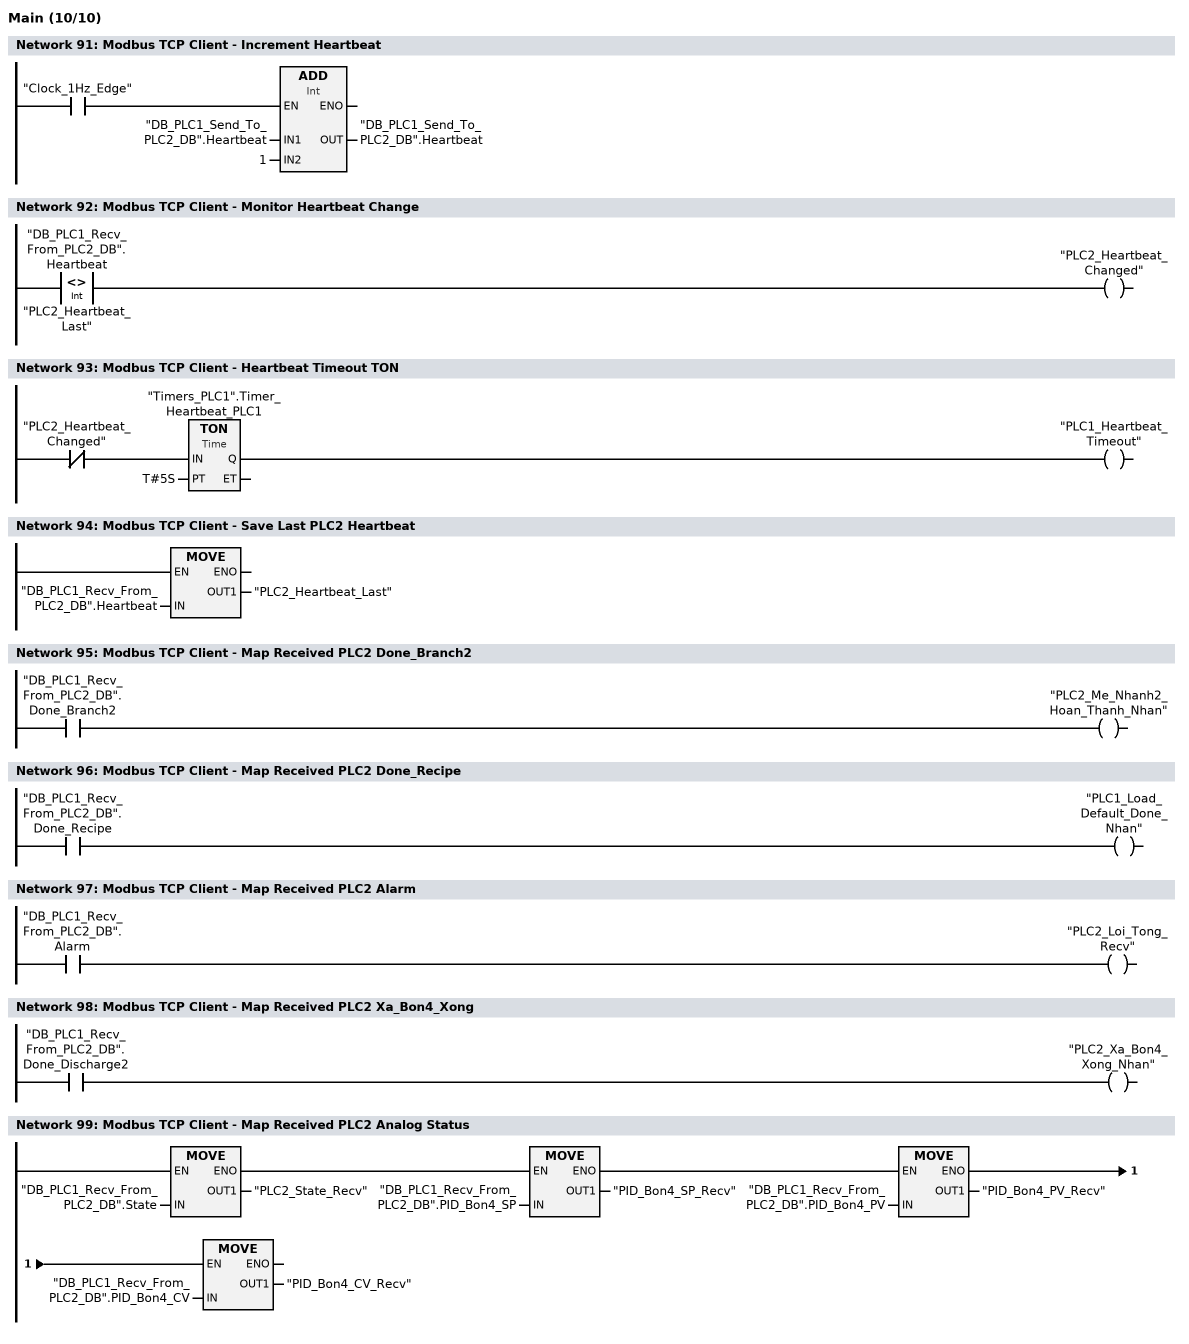
   RUNG wire#powerrail
      Contact( "Clock_1Hz_Edge" )
      { S7_Templates := "SrcType := Int"; S7_GenerateENO := "TRUE" } Add(in1 := "DB_PLC1_Send_To_PLC2_DB".Heartbeat, in2 := 1, out => "DB_PLC1_Send_To_PLC2_DB".Heartbeat)
   END_RUNG
   // the same network as SCL:
   IF "Clock_1Hz_Edge" THEN
       "DB_PLC1_Send_To_PLC2_DB".Heartbeat := "DB_PLC1_Send_To_PLC2_DB".Heartbeat + 1;
   END_IF;
END_REGION

REGION Network 92: Modbus TCP Client - Monitor Heartbeat Change
   RUNG wire#powerrail
      { S7_Templates := "SrcType := Int" } NE_Contact(in1 := "DB_PLC1_Recv_From_PLC2_DB".Heartbeat, in2 := "PLC2_Heartbeat_Last")
      Coil( "PLC2_Heartbeat_Changed" )
   END_RUNG
   // the same network as SCL:
   "PLC2_Heartbeat_Changed" := "DB_PLC1_Recv_From_PLC2_DB".Heartbeat <> "PLC2_Heartbeat_Last";
END_REGION

REGION Network 93: Modbus TCP Client - Heartbeat Timeout TON
   RUNG wire#powerrail
      I_Contact( "PLC2_Heartbeat_Changed" )
      { S7_Templates := "time_type := Time" } "Timers_PLC1".Timer_Heartbeat_PLC1.TON(pt := T#5S, et =>)
      Coil( "PLC1_Heartbeat_Timeout" )
   END_RUNG
   // the same network as SCL:
   "Timers_PLC1".Timer_Heartbeat_PLC1.TON(IN := NOT "PLC2_Heartbeat_Changed", PT := T#5S);
   "PLC1_Heartbeat_Timeout" := "Timers_PLC1".Timer_Heartbeat_PLC1.Q;
END_REGION

REGION Network 94: Modbus TCP Client - Save Last PLC2 Heartbeat
   RUNG wire#powerrail
      { S7_GenerateENO := "TRUE" } Move(in := "DB_PLC1_Recv_From_PLC2_DB".Heartbeat, out1 => "PLC2_Heartbeat_Last")
   END_RUNG
   // the same network as SCL:
   "PLC2_Heartbeat_Last" := "DB_PLC1_Recv_From_PLC2_DB".Heartbeat;
END_REGION

REGION Network 95: Modbus TCP Client - Map Received PLC2 Done_Branch2
   RUNG wire#powerrail
      Contact( "DB_PLC1_Recv_From_PLC2_DB".Done_Branch2 )
      Coil( "PLC2_Me_Nhanh2_Hoan_Thanh_Nhan" )
   END_RUNG
   // the same network as SCL:
   "PLC2_Me_Nhanh2_Hoan_Thanh_Nhan" := "DB_PLC1_Recv_From_PLC2_DB".Done_Branch2;
END_REGION

REGION Network 96: Modbus TCP Client - Map Received PLC2 Done_Recipe
   RUNG wire#powerrail
      Contact( "DB_PLC1_Recv_From_PLC2_DB".Done_Recipe )
      Coil( "PLC1_Load_Default_Done_Nhan" )
   END_RUNG
   // the same network as SCL:
   "PLC1_Load_Default_Done_Nhan" := "DB_PLC1_Recv_From_PLC2_DB".Done_Recipe;
END_REGION

REGION Network 97: Modbus TCP Client - Map Received PLC2 Alarm
   RUNG wire#powerrail
      Contact( "DB_PLC1_Recv_From_PLC2_DB".Alarm )
      Coil( "PLC2_Loi_Tong_Recv" )
   END_RUNG
   // the same network as SCL:
   "PLC2_Loi_Tong_Recv" := "DB_PLC1_Recv_From_PLC2_DB".Alarm;
END_REGION

REGION Network 98: Modbus TCP Client - Map Received PLC2 Xa_Bon4_Xong
   RUNG wire#powerrail
      Contact( "DB_PLC1_Recv_From_PLC2_DB".Done_Discharge2 )
      Coil( "PLC2_Xa_Bon4_Xong_Nhan" )
   END_RUNG
   // the same network as SCL:
   "PLC2_Xa_Bon4_Xong_Nhan" := "DB_PLC1_Recv_From_PLC2_DB".Done_Discharge2;
END_REGION

REGION Network 99: Modbus TCP Client - Map Received PLC2 Analog Status
   RUNG wire#powerrail
      { S7_GenerateENO := "TRUE" } Move(in := "DB_PLC1_Recv_From_PLC2_DB".State, out1 => "PLC2_State_Recv")
      { S7_GenerateENO := "TRUE" } Move(in := "DB_PLC1_Recv_From_PLC2_DB".PID_Bon4_SP, out1 => "PID_Bon4_SP_Recv")
      { S7_GenerateENO := "TRUE" } Move(in := "DB_PLC1_Recv_From_PLC2_DB".PID_Bon4_PV, out1 => "PID_Bon4_PV_Recv")
      { S7_GenerateENO := "TRUE" } Move(in := "DB_PLC1_Recv_From_PLC2_DB".PID_Bon4_CV, out1 => "PID_Bon4_CV_Recv")
   END_RUNG
   // the same network as SCL:
   // ENO of a box is taken as its EN; it also drops when the box reports an error
   "PLC2_State_Recv" := "DB_PLC1_Recv_From_PLC2_DB".State;
   "PID_Bon4_SP_Recv" := "DB_PLC1_Recv_From_PLC2_DB".PID_Bon4_SP;
   "PID_Bon4_PV_Recv" := "DB_PLC1_Recv_From_PLC2_DB".PID_Bon4_PV;
   "PID_Bon4_CV_Recv" := "DB_PLC1_Recv_From_PLC2_DB".PID_Bon4_CV;
END_REGION
END_ORGANIZATION_BLOCK
